TYPE MaxString : STRING(255); END_TYPE

(* stored: Version 1.1.0.1, ProductVersion 3.1.4022.7
   DUT MaxString: Id {24fb4e5b-aefa-4bdd-8414-9e6a91f82571} *)
